TEXTLIST InputText
  0 = 'IN00 启动' | Chinese: 'IN00 启动' | English: 'IN00 bStart' | Vietnamese: 'IN00 Khởi động'
  1 = 'IN01 停止' | Chinese: 'IN01 停止' | English: 'IN01 bStop' | Vietnamese: 'IN01 Dừng lại'
  2 = 'IN02 报警复位' | Chinese: 'IN02 报警复位' | English: 'IN02 bResetAlarm' | Vietnamese: 'IN02 Báo động thiết lập lại'
  3 = 'IN03 急停' | Chinese: 'IN03 急停' | English: 'IN03 bEStop' | Vietnamese: 'IN03 Vội dừng lại'
  4 = 'IN04 安全门开关' | Chinese: 'IN04 安全门开关' | English: 'IN04 bDoor' | Vietnamese: 'IN04 Chuyển đổi cửa an toàn'
  5 = 'IN05 预留' | Chinese: 'IN05 预留' | English: 'IN05 bNone1' | Vietnamese: 'IN05 Dành riêng'
  6 = 'IN06 预留' | Chinese: 'IN06 预留' | English: 'IN06 bNone2' | Vietnamese: 'IN06 Dành riêng'
  7 = 'IN07 主流线分料气缸原位(缩回)' | Chinese: 'IN07 主流线分料气缸原位(缩回)' | English: 'IN07 bLine0Part_Cyl_H' | Vietnamese: 'IN07 Xi lanh phân phối dòng chính'
  8 = 'IN08 主流线分料气缸工作位(伸出)' | Chinese: 'IN08 主流线分料气缸工作位(伸出)' | English: 'IN08 bLine0Part_Cyl_W' | Vietnamese: 'IN08 Xi lanh làm việc dòng chính'
  9 = 'IN09 主流线阻挡气缸原位(缩回)' | Chinese: 'IN09 主流线阻挡气缸原位(缩回)' | English: 'IN09 bLine0Prevent_Cyl_H' | Vietnamese: 'IN09 Dòng chính chặn xi lanh'
  10 = 'IN0A 主流线阻挡气缸工作位(伸出)' | Chinese: 'IN0A 主流线阻挡气缸工作位(伸出)' | English: 'IN0A bLine0Prevent_Cyl_W' | Vietnamese: 'IN0A Dòng chính chặn vị trí làm việc của xi lanh'
  11 = 'IN0B 流水线1提升气缸原位(下降)' | Chinese: 'IN0B 流水线1提升气缸原位(下降)' | English: 'IN0B bLine1Elevator_Cyl_H' | Vietnamese: 'IN0B Xi lanh nâng cấp trong dòng 1'
  12 = 'IN0C 流水线1提升气缸工作位(上升)' | Chinese: 'IN0C 流水线1提升气缸工作位(上升)' | English: 'IN0C bLine1Elevator_Cyl_W' | Vietnamese: 'IN0C Xi lanh làm việc 1 nâng cấp đường ống'
  13 = 'IN0D 流水线1顶升气缸原位(缩回)' | Chinese: 'IN0D 流水线1顶升气缸原位(缩回)' | English: 'IN0D bLine1Lift_Cyl_H' | Vietnamese: 'IN0D Xi lanh 1 lít trong đường ống'
  14 = 'IN0E 流水线1顶升气缸工作位(伸出)' | Chinese: 'IN0E 流水线1顶升气缸工作位(伸出)' | English: 'IN0E bLine1Lift_Cyl_W' | Vietnamese: 'IN0E Xi lanh làm việc 1 lít dây chuyền sản xuất'
  15 = 'IN0F 流水线1阻挡气缸原位(缩回)' | Chinese: 'IN0F 流水线1阻挡气缸原位(缩回)' | English: 'IN0F bLine1Prevent_Cyl_H' | Vietnamese: 'IN0F Dòng 1 ngăn xi lanh vị trí'
  16 = 'IN10 流水线1阻挡气缸工作位(伸出)' | Chinese: 'IN10 流水线1阻挡气缸工作位(伸出)' | English: 'IN10 bLine1Prevent_Cyl_W' | Vietnamese: 'IN10 Dây chuyền sản xuất 1 ngăn xi lanh vị trí làm việc'
  17 = 'IN11 流水线1旋转气缸原位' | Chinese: 'IN11 流水线1旋转气缸原位' | English: 'IN11 bLine1Rotate_Cyl_H' | Vietnamese: 'IN11 Xi lanh xoay dòng 1 vị trí'
  18 = 'IN12 流水线1旋转气缸工作位' | Chinese: 'IN12 流水线1旋转气缸工作位' | English: 'IN12 bLine1Rotate_Cyl_W' | Vietnamese: 'IN12 Xi lanh quay dòng 1 vị trí làm việc'
  19 = 'IN13 流水线1调宽气缸原位1(张开)' | Chinese: 'IN13 流水线1调宽气缸原位1(张开)' | English: 'IN13 bLine1Adjust1_Cyl_H' | Vietnamese: 'IN13 Dây chuyền sản xuất 1 mở rộng xi lanh ở vị trí 1'
  20 = 'IN14 流水线1调宽气缸工作位1(夹紧)' | Chinese: 'IN14 流水线1调宽气缸工作位1(夹紧)' | English: 'IN14 bLine1Adjust1_Cyl_W' | Vietnamese: 'IN14 Xi lanh làm việc 1 mở rộng dòng 1'
  21 = 'IN15 流水线1调宽气缸原位2(张开)' | Chinese: 'IN15 流水线1调宽气缸原位2(张开)' | English: 'IN15 bLine1Adjust2_Cyl_H' | Vietnamese: 'IN15 Xi lanh ở vị trí 2 mở rộng dòng 1'
  22 = 'IN16 流水线1调宽气缸工作位2(夹紧)' | Chinese: 'IN16 流水线1调宽气缸工作位2(夹紧)' | English: 'IN16 bLine1Adjust2_Cyl_W' | Vietnamese: 'IN16 Dây chuyền sản xuất 1 mở xi lanh làm việc 2'
  23 = 'IN17 流水线2顶升气缸原位(缩回)' | Chinese: 'IN17 流水线2顶升气缸原位(缩回)' | English: 'IN17 bLine2Lift_Cyl_H' | Vietnamese: 'IN17 Dây chuyền sản xuất 2 lít xi lanh vị trí'
  24 = 'IN18 流水线2顶升气缸工作位(伸出)' | Chinese: 'IN18 流水线2顶升气缸工作位(伸出)' | English: 'IN18 bLine2Lift_Cyl_W' | Vietnamese: 'IN18 Dây chuyền sản xuất 2 lít xi lanh vị trí'
  25 = 'IN19 流水线2阻挡气缸原位(缩回)' | Chinese: 'IN19 流水线2阻挡气缸原位(缩回)' | English: 'IN19 bLine2Prevent_Cyl_H' | Vietnamese: 'IN19 Dây chuyền sản xuất 2 chặn xi lanh vị trí'
  26 = 'IN1A 流水线2阻挡气缸工作位(伸出)' | Chinese: 'IN1A 流水线2阻挡气缸工作位(伸出)' | English: 'IN1A bLine2Prevent_Cyl_W' | Vietnamese: 'IN1A Dây chuyền sản xuất 2 ngăn xi lanh vị trí làm việc'
  27 = 'IN1B 流水线2校平气缸1原位(缩回)' | Chinese: 'IN1B 流水线2校平气缸1原位(缩回)' | English: 'IN1B bLine2Standard1_Cyl_H' | Vietnamese: 'IN1B Dòng 2 cân bằng xi lanh 1 tại chỗ'
  28 = 'IN1C 流水线2校平气缸1工作位(伸出)' | Chinese: 'IN1C 流水线2校平气缸1工作位(伸出)' | English: 'IN1C bLine2Standard1_Cyl_W' | Vietnamese: 'IN1C Dòng 2 cân bằng xi lanh 1 vị trí'
  29 = 'IN1D 流水线2校平气缸2原位(缩回)' | Chinese: 'IN1D 流水线2校平气缸2原位(缩回)' | English: 'IN1D bLine2Standard2_Cyl_H' | Vietnamese: 'IN1D Dòng 2 cân bằng xi lanh 2 vị trí'
  30 = 'IN1E 流水线2校平气缸2工作位(伸出)' | Chinese: 'IN1E 流水线2校平气缸2工作位(伸出)' | English: 'IN1E bLine2Standard2_Cyl_W' | Vietnamese: 'IN1E Dòng 2 cân bằng xi lanh 2 vị trí'
  31 = 'IN1F 流水线2解锁侧推气缸1原位(缩回)' | Chinese: 'IN1F 流水线2解锁侧推气缸1原位(缩回)' | English: 'IN1F bLine2OpenLateral1_Cyl_H' | Vietnamese: 'IN1F Dây chuyền sản xuất 2 mở khóa xi lanh bên đẩy 1 vị trí'
  32 = 'IN20 流水线2解锁侧推气缸1工作位(伸出)' | Chinese: 'IN20 流水线2解锁侧推气缸1工作位(伸出)' | English: 'IN20 bLine2OpenLateral1_Cyl_W' | Vietnamese: 'IN20 Dây chuyền sản xuất 2 mở khóa bên đẩy xi lanh 1 vị trí'
  33 = 'IN21 流水线2解锁旋转气缸原位(左位)' | Chinese: 'IN21 流水线2解锁旋转气缸原位(左位)' | English: 'IN21 bLine2OpenRotate_Cyl_H' | Vietnamese: 'IN21 Dòng 2 mở khóa xi lanh quay vị trí'
  34 = 'IN22 流水线2解锁旋转气缸工作位(右位)' | Chinese: 'IN22 流水线2解锁旋转气缸工作位(右位)' | English: 'IN22 bLine2OpenRotate_Cyl_W' | Vietnamese: 'IN22 Dây chuyền sản xuất 2 mở khóa xi lanh quay vị trí làm việc'
  35 = 'IN23 流水线2解锁侧推气缸2原位(缩回)' | Chinese: 'IN23 流水线2解锁侧推气缸2原位(缩回)' | English: 'IN23 bLine2OpenLateral2_Cyl_H' | Vietnamese: 'IN23 Dòng 2 mở khóa bên đẩy xi lanh 2 vị trí'
  36 = 'IN24 流水线2解锁侧推气缸2工作位(伸出)' | Chinese: 'IN24 流水线2解锁侧推气缸2工作位(伸出)' | English: 'IN24 bLine2OpenLateral2_Cyl_W' | Vietnamese: 'IN24 Dây chuyền sản xuất 2 mở khóa bên đẩy xi lanh 2 vị trí'
  37 = 'IN25 空' | Chinese: 'IN25 空' | English: 'IN25 None' | Vietnamese: 'IN25 trống'
  38 = 'IN26 空' | Chinese: 'IN26 空' | English: 'IN26 None1' | Vietnamese: 'IN26 trống'
  39 = 'IN27 流水线3上料位顶升原位(缩回)' | Chinese: 'IN27 流水线3上料位顶升原位(缩回)' | English: 'IN27 bLine3LoadLift_Cyl_H' | Vietnamese: 'IN27 Dòng 3 lên vị trí'
  40 = 'IN28 流水线3上料位顶升工作位(伸出)' | Chinese: 'IN28 流水线3上料位顶升工作位(伸出)' | English: 'IN28 bLine3LoadLift_Cyl_W' | Vietnamese: 'IN28 Dây chuyền sản xuất 3 lên vị trí'
  41 = 'IN29 流水线3上料位阻挡原位(缩回)' | Chinese: 'IN29 流水线3上料位阻挡原位(缩回)' | English: 'IN29 bLine3LoadPrevent_Cyl_H' | Vietnamese: 'IN29 Dòng 3 lên cấp độ để ngăn chặn vị trí'
  42 = 'IN2A 流水线3上料位阻挡工作位(伸出)' | Chinese: 'IN2A 流水线3上料位阻挡工作位(伸出)' | English: 'IN2A bLine3LoadPrevent_Cyl_W' | Vietnamese: 'IN2A Dòng 3 lên vị trí công việc'
  43 = 'IN2B 流水线3上料位旋转原位' | Chinese: 'IN2B 流水线3上料位旋转原位' | English: 'IN2B bLine3LoadRotate_Cyl_H' | Vietnamese: 'IN2B Dòng 3 cấp độ quay vị trí'
  44 = 'IN2C 流水线3上料位旋转工作位' | Chinese: 'IN2C 流水线3上料位旋转工作位' | English: 'IN2C bLine3LoadRotate_Cyl_W' | Vietnamese: 'IN2C Dây chuyền sản xuất 3 vị trí quay'
  45 = 'IN2D 流水线3解锁位顶升原位(缩回)' | Chinese: 'IN2D 流水线3解锁位顶升原位(缩回)' | English: 'IN2D bLine3OpenLift_Cyl_H' | Vietnamese: 'IN2D Dòng 3 mở khóa vị trí nâng cao vị trí'
  46 = 'IN2E 流水线3解锁位顶升工作位(伸出)' | Chinese: 'IN2E 流水线3解锁位顶升工作位(伸出)' | English: 'IN2E bLine3OpenLift_Cyl_W' | Vietnamese: 'IN2E Dòng 3 mở khóa lên vị trí làm việc'
  47 = 'IN2F 流水线3解锁位阻挡原位(缩回)' | Chinese: 'IN2F 流水线3解锁位阻挡原位(缩回)' | English: 'IN2F bLine3OpenPrevent_Cyl_H' | Vietnamese: 'IN2F Dòng 3 mở khóa vị trí để ngăn vị trí'
  48 = 'IN30 流水线3解锁位阻挡工作位(伸出)' | Chinese: 'IN30 流水线3解锁位阻挡工作位(伸出)' | English: 'IN30 bLine3OpenPrevent_Cyl_W' | Vietnamese: 'IN30 Dòng 3 mở khóa vị trí làm việc'
  49 = 'IN31 流水线3校平气缸1原位(缩回)' | Chinese: 'IN31 流水线3校平气缸1原位(缩回)' | English: 'IN31 bLine3Standard1_Cyl_H' | Vietnamese: 'IN31 Dòng 3 phẳng xi lanh 1 vị trí'
  50 = 'IN32 流水线3校平气缸1工作位(伸出)' | Chinese: 'IN32 流水线3校平气缸1工作位(伸出)' | English: 'IN32 bLine3Standard1_Cyl_W' | Vietnamese: 'IN32 Dòng 3 cân bằng xi lanh 1 vị trí'
  51 = 'IN33 流水线3校平气缸2原位(缩回)' | Chinese: 'IN33 流水线3校平气缸2原位(缩回)' | English: 'IN33 bLine3Standard2_Cyl_H' | Vietnamese: 'IN33 Dòng 3 cân bằng xi lanh 2 vị trí'
  52 = 'IN34 流水线3校平气缸2工作位(伸出)' | Chinese: 'IN34 流水线3校平气缸2工作位(伸出)' | English: 'IN34 bLine3Standard2_Cyl_W' | Vietnamese: 'IN34 Dòng 3 cân bằng xi lanh 2 vị trí'
  53 = 'IN35 流水线3解锁侧推气缸1原位(缩回)' | Chinese: 'IN35 流水线3解锁侧推气缸1原位(缩回)' | English: 'IN35 bLine3OpenLateral1_Cyl_H' | Vietnamese: 'IN35 Dòng 3 mở khóa bên đẩy xi lanh 1 vị trí'
  54 = 'IN36 流水线3解锁侧推气缸1工作位(伸出)' | Chinese: 'IN36 流水线3解锁侧推气缸1工作位(伸出)' | English: 'IN36 bLine3OpenLateral1_Cyl_W' | Vietnamese: 'IN36 Dây chuyền sản xuất 3 mở khóa xi lanh bên đẩy 1 vị trí'
  55 = 'IN37 流水线3解锁旋转气缸原位(左位)' | Chinese: 'IN37 流水线3解锁旋转气缸原位(左位)' | English: 'IN37 bLine3OpenRotate_Cyl_H' | Vietnamese: 'IN37 Dòng 3 mở khóa xi lanh quay vị trí'
  56 = 'IN38 流水线3解锁旋转气缸工作位(右位)' | Chinese: 'IN38 流水线3解锁旋转气缸工作位(右位)' | English: 'IN38 bLine3OpenRotate_Cyl_W' | Vietnamese: 'IN38 Dây chuyền sản xuất 3 mở khóa xi lanh quay vị trí làm việc'
  57 = 'IN39 流水线3解锁侧推气缸2原位(缩回)' | Chinese: 'IN39 流水线3解锁侧推气缸2原位(缩回)' | English: 'IN39 bLine3OpenLateral2_Cyl_H' | Vietnamese: 'IN39 Dòng 3 mở khóa bên đẩy xi lanh 2 vị trí'
  58 = 'IN3A 流水线3解锁侧推气缸2工作位(伸出)' | Chinese: 'IN3A 流水线3解锁侧推气缸2工作位(伸出)' | English: 'IN3A bLine3OpenLateral2_Cyl_W' | Vietnamese: 'IN3A Dòng 3 mở khóa bên đẩy xi lanh 2 vị trí'
  59 = 'IN3B 空' | Chinese: 'IN3B 空' | English: 'IN3B None3' | Vietnamese: 'IN3B trống'
  60 = 'IN3C 空' | Chinese: 'IN3C 空' | English: 'IN3C None4' | Vietnamese: 'IN3C trống'
  61 = 'IN3D 取料模组升降气缸1原位(上升)' | Chinese: 'IN3D 取料模组升降气缸1原位(上升)' | English: 'IN3D bTakeLift1_Cyl_H' | Vietnamese: 'IN3D Lấy khối nâng xi lanh 1 vị trí'
  62 = 'IN3E 取料模组升降气缸1工作位(下降)' | Chinese: 'IN3E 取料模组升降气缸1工作位(下降)' | English: 'IN3E bTakeLift1_Cyl_W' | Vietnamese: 'IN3E Lấy khối nâng xi lanh 1 vị trí'
  63 = 'IN3F 取料模组升降气缸2原位(上升)' | Chinese: 'IN3F 取料模组升降气缸2原位(上升)' | English: 'IN3F bTakeLift2_Cyl_H' | Vietnamese: 'IN3F Lấy khối nâng xi lanh 2 vị trí'
  64 = 'IN40 取料模组升降气缸2工作位(下降)' | Chinese: 'IN40 取料模组升降气缸2工作位(下降)' | English: 'IN40 bTakeLift2_Cyl_W' | Vietnamese: 'IN40 Chế độ nâng xi lanh 2 làm việc'
  65 = 'IN41 取料模组夹紧气缸原位(张开)' | Chinese: 'IN41 取料模组夹紧气缸原位(张开)' | English: 'IN41 bTakeClamp_Cyl_H' | Vietnamese: 'IN41 Lấy mô-đun kẹp xi lanh vị trí'
  66 = 'IN42 取料模组夹紧气缸工作位(夹紧)' | Chinese: 'IN42 取料模组夹紧气缸工作位(夹紧)' | English: 'IN42 bTakeClamp_Cyl_W' | Vietnamese: 'IN42 Lấy mô-đun kẹp xi lanh vị trí làm việc'
  67 = 'IN43 下UC模组升降气缸原位(上升)' | Chinese: 'IN43 下UC模组升降气缸原位(上升)' | English: 'IN43 bUcLift_Cyl_H' | Vietnamese: 'IN43 Xi lanh nâng theo mô-đun UC'
  68 = 'IN44 下UC模组升降气缸工作位(下降)' | Chinese: 'IN44 下UC模组升降气缸工作位(下降)' | English: 'IN44 bUcLift_Cyl_W' | Vietnamese: 'IN44 Xi lanh nâng theo mô-đun UC'
  69 = 'IN45 下UC模组夹紧气缸原位(张开)' | Chinese: 'IN45 下UC模组夹紧气缸原位(张开)' | English: 'IN45 bUcClamp_Cyl_H' | Vietnamese: 'IN45 Mô-đun dưới UC kẹp xi lanh vào vị trí'
  70 = 'IN46 下UC模组夹紧气缸工作位(夹紧)' | Chinese: 'IN46 下UC模组夹紧气缸工作位(夹紧)' | English: 'IN46 bUcClamp_Cyl_W' | Vietnamese: 'IN46 Mô-đun dưới UC kẹp xi lanh vị trí làm việc'
  71 = 'IN47 下UC模组摆动气缸原位(上升)' | Chinese: 'IN47 下UC模组摆动气缸原位(上升)' | English: 'IN47 bUcSwing_Cyl_H' | Vietnamese: 'IN47 Mô-đun dưới UC đang chuyển động xi lanh'
  72 = 'IN48 下UC模组摆动气缸工作位(下降)' | Chinese: 'IN48 下UC模组摆动气缸工作位(下降)' | English: 'IN48 bUcSwing_Cyl_W' | Vietnamese: 'IN48 Mô-đun dưới UC đu vị trí xi lanh'
  73 = 'IN49 下UC升降气缸1原位(下降)' | Chinese: 'IN49 下UC升降气缸1原位(下降)' | English: 'IN49 bUcLift1_Cyl_H' | Vietnamese: 'IN49 Xi lanh nâng UC 1 đang ở vị trí'
  74 = 'IN4A 下UC升降气缸1工作位(上升)' | Chinese: 'IN4A 下UC升降气缸1工作位(上升)' | English: 'IN4A bUcLift1_Cyl_W' | Vietnamese: 'IN4A Xi lanh nâng dưới UC 1 vị trí'
  75 = 'IN4B 下UC夹紧气缸1原位(张开)' | Chinese: 'IN4B 下UC夹紧气缸1原位(张开)' | English: 'IN4B bUcClamp1_Cyl_H' | Vietnamese: 'IN4B Khóa xi lanh 1 lại'
  76 = 'IN4C 下UC夹紧气缸1工作位(夹紧)' | Chinese: 'IN4C 下UC夹紧气缸1工作位(夹紧)' | English: 'IN4C bUcClamp1_Cyl_W' | Vietnamese: 'IN4C Khóa xi lanh 1 lại'
  77 = 'IN4D 下UC旋转气缸1原位(右位)' | Chinese: 'IN4D 下UC旋转气缸1原位(右位)' | English: 'IN4D bUcRotate1_Cyl_H' | Vietnamese: 'IN4D Xi lanh quay dưới UC đang ở vị trí 1'
  78 = 'IN4E 下UC旋转气缸1工作位(左位)' | Chinese: 'IN4E 下UC旋转气缸1工作位(左位)' | English: 'IN4E bUcRotate1_Cyl_W' | Vietnamese: 'IN4E Xi lanh quay dưới UC đang hoạt động'
  79 = 'IN4F 下UC升降气缸2原位(下降)' | Chinese: 'IN4F 下UC升降气缸2原位(下降)' | English: 'IN4F bUcLift2_Cyl_H' | Vietnamese: 'IN4F Xi lanh nâng UC 2 vị trí'
  80 = 'IN50 下UC升降气缸2工作位(上升)' | Chinese: 'IN50 下UC升降气缸2工作位(上升)' | English: 'IN50 bUcLift2_Cyl_W' | Vietnamese: 'IN50 Xi lanh nâng dưới UC 2 vị trí'
  81 = 'IN51 下UC夹紧气缸2原位(张开)' | Chinese: 'IN51 下UC夹紧气缸2原位(张开)' | English: 'IN51 bUcClamp2_Cyl_H' | Vietnamese: 'IN51 Ống 2 đang ở vị trí'
  82 = 'IN52 下UC夹紧气缸2工作位(夹紧)' | Chinese: 'IN52 下UC夹紧气缸2工作位(夹紧)' | English: 'IN52 bUcClamp2_Cyl_W' | Vietnamese: 'IN52 Ống 2 đang hoạt động'
  83 = 'IN53 下UC旋转气缸2原位(右位)' | Chinese: 'IN53 下UC旋转气缸2原位(右位)' | English: 'IN53 bUcRotate2_Cyl_H' | Vietnamese: 'IN53 Xi lanh 2 quay dưới UC'
  84 = 'IN54 下UC旋转气缸2工作位(左位)' | Chinese: 'IN54 下UC旋转气缸2工作位(左位)' | English: 'IN54 bUcRotate2_Cyl_W' | Vietnamese: 'IN54 Xi lanh quay dưới UC đang hoạt động'
  85 = 'IN55 下UC皮带推料气缸原位(缩回)' | Chinese: 'IN55 下UC皮带推料气缸原位(缩回)' | English: 'IN55 bUcDrive_Cyl_H' | Vietnamese: 'IN55 Xi lanh đẩy dưới vành đai UC'
  86 = 'IN56 下UC皮带推料气缸工作位(伸出)' | Chinese: 'IN56 下UC皮带推料气缸工作位(伸出)' | English: 'IN56 bUcDrive_Cyl_W' | Vietnamese: 'IN56 Vị trí của xi lanh đẩy dưới vành đai UC'
  87 = 'IN57 下工装提升气缸1原位(下降)' | Chinese: 'IN57 下工装提升气缸1原位(下降)' | English: 'IN57 bFrockElevator1_Cyl_H' | Vietnamese: 'IN57 Máy nâng xi lanh 1 vị trí'
  88 = 'IN58 下工装提升气缸1工作位(上升)' | Chinese: 'IN58 下工装提升气缸1工作位(上升)' | English: 'IN58 bFrockElevator1_Cyl_W' | Vietnamese: 'IN58 Máy nâng xi lanh 1 vị trí'
  89 = 'IN59 下工装旋转压紧气缸1原位(缩回)' | Chinese: 'IN59 下工装旋转压紧气缸1原位(缩回)' | English: 'IN59 bFrockRotateDown1_Cyl_H' | Vietnamese: 'IN59 Tải trọng xoay xi lanh 1 vị trí'
  90 = 'IN5A 下工装旋转压紧气缸1工作位(伸出)' | Chinese: 'IN5A 下工装旋转压紧气缸1工作位(伸出)' | English: 'IN5A bFrockRotateDown1_Cyl_W' | Vietnamese: 'IN5A Xi lanh xoay ép xi lanh 1 vị trí làm việc'
  91 = 'IN5B 下工装拨料气缸1原位(缩回)' | Chinese: 'IN5B 下工装拨料气缸1原位(缩回)' | English: 'IN5B bFrockPush1_Cyl_H' | Vietnamese: 'IN5B Xi lanh 1 tải trọng'
  92 = 'IN5C 下工装拨料气缸1工作位(伸出)' | Chinese: 'IN5C 下工装拨料气缸1工作位(伸出)' | English: 'IN5C bFrockPush1_Cyl_W' | Vietnamese: 'IN5C Xi lanh công cụ đo 1 vị trí'
  93 = 'IN5D 下工装提升气缸2原位(下降)' | Chinese: 'IN5D 下工装提升气缸2原位(下降)' | English: 'IN5D bFrockElevator2_Cyl_H' | Vietnamese: 'IN5D Máy nâng xi lanh 2 vị trí'
  94 = 'IN5E 下工装提升气缸2工作位(上升)' | Chinese: 'IN5E 下工装提升气缸2工作位(上升)' | English: 'IN5E bFrockElevator2_Cyl_W' | Vietnamese: 'IN5E Máy nâng xi lanh 2 vị trí'
  95 = 'IN5F 下工装旋转压紧气缸2原位(缩回)' | Chinese: 'IN5F 下工装旋转压紧气缸2原位(缩回)' | English: 'IN5F bFrockRotateDown2_Cyl_H' | Vietnamese: 'IN5F Tải trọng xoay xi lanh 2 trong vị trí'
  96 = 'IN60 下工装旋转压紧气缸2工作位(伸出)' | Chinese: 'IN60 下工装旋转压紧气缸2工作位(伸出)' | English: 'IN60 bFrockRotateDown2_Cyl_W' | Vietnamese: 'IN60 Xi lanh xoay ép xi lanh 2 vị trí làm việc'
  97 = 'IN61 下工装拨料气缸2原位(缩回)' | Chinese: 'IN61 下工装拨料气缸2原位(缩回)' | English: 'IN61 bFrockPush2_Cyl_H' | Vietnamese: 'IN61 Xi lanh theo tải trọng 2 vị trí'
  98 = 'IN62 下工装拨料气缸2工作位(伸出)' | Chinese: 'IN62 下工装拨料气缸2工作位(伸出)' | English: 'IN62 bFrockPush2_Cyl_W' | Vietnamese: 'IN62 Xi lanh xi lanh công cụ 2 vị trí'
  99 = 'IN63 下工装皮带推料气缸原位(缩回)' | Chinese: 'IN63 下工装皮带推料气缸原位(缩回)' | English: 'IN63 bFrockBelt_Cyl_H' | Vietnamese: 'IN63 Tải trọng vành đai đẩy xi lanh trong vị trí'
  100 = 'IN64 下工装皮带推料气缸工作位(伸出)' | Chinese: 'IN64 下工装皮带推料气缸工作位(伸出)' | English: 'IN64 bFrockBelt_Cyl_W' | Vietnamese: 'IN64 Dây chuyền đẩy xi lanh làm việc'
  101 = 'IN65 预留' | Chinese: 'IN65 预留' | English: 'IN65 bNone3' | Vietnamese: 'IN65 Dành riêng'
  102 = 'IN66 主流线分料光电' | Chinese: 'IN66 主流线分料光电' | English: 'IN66 bLine0Part' | Vietnamese: 'IN66 Dòng chính phân phối quang điện'
  103 = 'IN67 主流线阻挡光电' | Chinese: 'IN67 主流线阻挡光电' | English: 'IN67 bLine0Prevent' | Vietnamese: 'IN67 Dòng chính ngăn chặn quang điện'
  104 = 'IN68 主流线到位光电' | Chinese: 'IN68 主流线到位光电' | English: 'IN68 bLine0Place' | Vietnamese: 'IN68 Dòng chính vào vị trí quang điện'
  105 = 'IN69 流水线1流入光电' | Chinese: 'IN69 流水线1流入光电' | English: 'IN69 bLine1PalletCheck1' | Vietnamese: 'IN69 Dòng 1 chảy vào quang điện'
  106 = 'IN6A 流水线1到位光电' | Chinese: 'IN6A 流水线1到位光电' | English: 'IN6A bLine1PalletCheck2' | Vietnamese: 'IN6A Lắp ráp 1 vị trí quang điện'
  107 = 'IN6B 流水线1流出光电' | Chinese: 'IN6B 流水线1流出光电' | English: 'IN6B bLine1PalletCheck3' | Vietnamese: 'IN6B Dòng 1 ra khỏi quang điện'
  108 = 'IN6C 流水线2流入光电' | Chinese: 'IN6C 流水线2流入光电' | English: 'IN6C bLine2PalletCheck1' | Vietnamese: 'IN6C Dòng 2 chảy vào quang điện'
  109 = 'IN6D 流水线2到位光电' | Chinese: 'IN6D 流水线2到位光电' | English: 'IN6D bLine2PalletCheck2' | Vietnamese: 'IN6D Lắp ráp 2 vị trí quang điện'
  110 = 'IN6E 流水线2流出光电' | Chinese: 'IN6E 流水线2流出光电' | English: 'IN6E bLine2PalletCheck3' | Vietnamese: 'IN6E Dòng 2 ra khỏi quang điện'
  111 = 'IN6F 流水线3上料位流入光电' | Chinese: 'IN6F 流水线3上料位流入光电' | English: 'IN6F bLine3PalletCheck1' | Vietnamese: 'IN6F Dòng 3 cấp nạp vào optoelectronics'
  112 = 'IN70 流水线3上料位到位光电' | Chinese: 'IN70 流水线3上料位到位光电' | English: 'IN70 bLine3PalletCheck2' | Vietnamese: 'IN70 Dòng 3 lên vị trí quang điện'
  113 = 'IN71 流水线3上料位流出光电' | Chinese: 'IN71 流水线3上料位流出光电' | English: 'IN71 bLine3PalletCheck3' | Vietnamese: 'IN71 Dòng 3 lên máy phát điện'
  114 = 'IN72 流水线3解锁位流入光电' | Chinese: 'IN72 流水线3解锁位流入光电' | English: 'IN72 bLine3OpenCheck1' | Vietnamese: 'IN72 Dây chuyền sản xuất 3 ổ khóa vào optoelectronics'
  115 = 'IN73 流水线3解锁位到位光电' | Chinese: 'IN73 流水线3解锁位到位光电' | English: 'IN73 bLine3OpenCheck2' | Vietnamese: 'IN73 Dòng 3 mở khóa vị trí quang điện'
  116 = 'IN74 流水线3解锁位流出光电' | Chinese: 'IN74 流水线3解锁位流出光电' | English: 'IN74 bLine3OpenCheck3' | Vietnamese: 'IN74 Dòng 3 mở khóa vị trí ra khỏi optoelectronics'
  117 = 'IN75 下UC模组UC有无检测1' | Chinese: 'IN75 下UC模组UC有无检测1' | English: 'IN75 bUcCheck1' | Vietnamese: 'IN75 Mô-đun UC dưới UC không có phát hiện 1'
  118 = 'IN76 下UC皮带UC有无检测2' | Chinese: 'IN76 下UC皮带UC有无检测2' | English: 'IN76 bUcCheck2' | Vietnamese: 'IN76 Dưới vành đai UC không có phát hiện 2'
  119 = 'IN77 下UC皮带UC有无检测3' | Chinese: 'IN77 下UC皮带UC有无检测3' | English: 'IN77 bUcCheck3' | Vietnamese: 'IN77 Dưới vành đai UC UC không có phát hiện 3'
  120 = 'IN78 下UC皮带到位检测' | Chinese: 'IN78 下UC皮带到位检测' | English: 'IN78 bUcBeltDone' | Vietnamese: 'IN78 Xác định vị trí của cảnh sát chìm'
  121 = 'IN79 下UC皮带斜坡有无检测' | Chinese: 'IN79 下UC皮带斜坡有无检测' | English: 'IN79 bUcBeltNoneCheck' | Vietnamese: 'IN79 Không có phát hiện độ dốc dưới vành đai UC'
  122 = 'IN7A 下工装提升1工装有无检测' | Chinese: 'IN7A 下工装提升1工装有无检测' | English: 'IN7A bFrockElevator1NoneCheck' | Vietnamese: 'IN7A Công cụ nâng cấp 1 công cụ có là không có phát hiện'
  123 = 'IN7B 下工装提升2工装有无检测' | Chinese: 'IN7B 下工装提升2工装有无检测' | English: 'IN7B bFrockElevator2NoneCheck' | Vietnamese: 'IN7B Công cụ nâng cao 2 công cụ có là không có phát hiện'
  124 = 'IN7C 下工装皮带工装有无检测1' | Chinese: 'IN7C 下工装皮带工装有无检测1' | English: 'IN7C bFrockBeltNoneCheck1' | Vietnamese: 'IN7C Vành đai công việc không có không có phát hiện 1'
  125 = 'IN7D 下工装皮带工装有无检测2' | Chinese: 'IN7D 下工装皮带工装有无检测2' | English: 'IN7D bFrockBeltNoneCheck2' | Vietnamese: 'IN7D Vành đai công việc không có không có phát hiện 2'
  126 = 'IN7E 下工装皮带到位检测' | Chinese: 'IN7E 下工装皮带到位检测' | English: 'IN7E bFrockBeltDone' | Vietnamese: 'IN7E Thắt lưng ở vị trí'
  127 = 'IN7F 下工装皮带斜坡有无检测' | Chinese: 'IN7F 下工装皮带斜坡有无检测' | English: 'IN7F bFrockBeltNoneCheck3' | Vietnamese: 'IN7F Công cụ vành đai dốc đã không được phát hiện'
   = ''
END_TEXTLIST

(* stored: Version 1.1.0.1, ProductVersion 3.1.4024.3
   TextList InputText: Id {a47183f6-45cc-4246-831a-883b90f1de4c} *)
